{attribute 'qualified_only'}
{attribute 'strict'}
TYPE E_FastDoorControlStates :
(
	INIT,
	IDLE,
	DOOR_UP,
	DOOR_DOWN
);
END_TYPE

(* stored: Version 1.1.0.1, ProductVersion 3.1.4024.9
   DUT E_FastDoorControlStates: Id {87ac8f8a-e611-4419-8470-e396440c2a46} *)
